% RSLogix 500 project DIAGNOSTICO_ML1400.RSS, saved by version 12.00.00.00 %
PROJECT "UNTITLED"    % processor: type code 64 %

PROGRAM FILES
  LAD 2   15 rungs

DATA FILES
  O0 OUTPUT  6 elements
  I1 INPUT  9 elements
  S2 STATUS  66 elements
  B3 BINARY  1 elements
  T4 TIMER  1 elements
  C5 COUNTER  1 elements
  R6 CONTROL  1 elements
  N7 INTEGER  20 elements
  F8 FLOAT  1 elements

LADDER 2
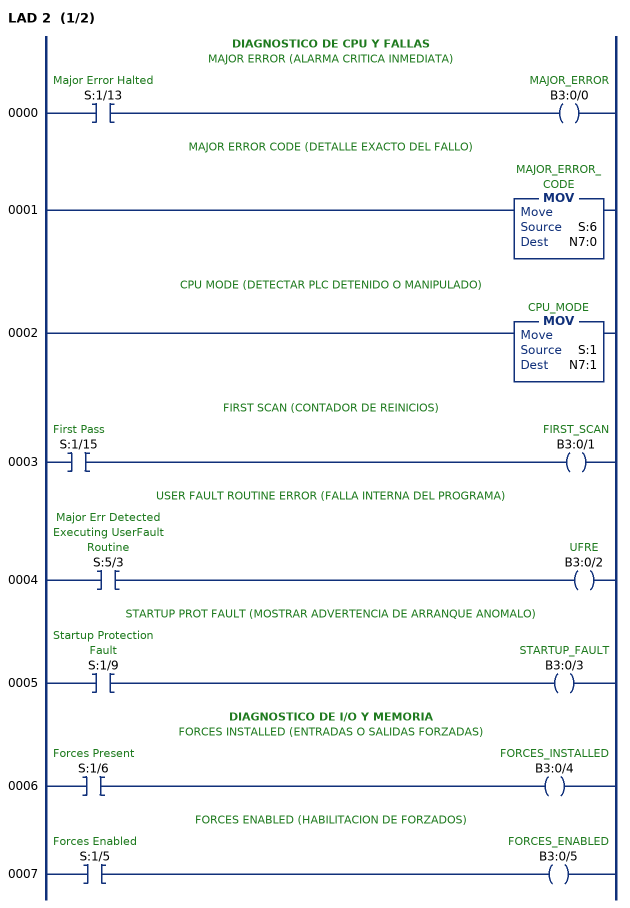
% Rung: 0 %
% TITLE: DIAGNOSTICO DE CPU Y FALLAS %
% MAJOR ERROR (ALARMA CRITICA INMEDIATA) %
SOR XIC S:1/13 OTE B3:0/0 EOR
%   S:1/13  "Major Error Halted" %
%   B3:0/0  MAJOR_ERROR %
% Rung: 1 %
% MAJOR ERROR CODE (DETALLE EXACTO DEL FALLO) %
SOR MOV S:6 N7:0 EOR
%   S:6  "Major Error Fault Code" %
%   N7:0  MAJOR_ERROR_CODE %
% Rung: 2 %
% CPU MODE (DETECTAR PLC DETENIDO O MANIPULADO) %
SOR MOV S:1 N7:1 EOR
%   S:1  "Processor Mode Status/ Control" %
%   N7:1  CPU_MODE %
% Rung: 3 %
% FIRST SCAN (CONTADOR DE REINICIOS) %
SOR XIC S:1/15 OTE B3:0/1 EOR
%   S:1/15  "First Pass" %
%   B3:0/1  FIRST_SCAN %
% Rung: 4 %
% USER FAULT ROUTINE ERROR (FALLA INTERNA DEL PROGRAMA) %
SOR XIC S:5/3 OTE B3:0/2 EOR
%   S:5/3  "Major Err Detected Executing UserFault Routine" %
%   B3:0/2  UFRE %
% Rung: 5 %
% STARTUP PROT FAULT (MOSTRAR ADVERTENCIA DE ARRANQUE ANOMALO) %
SOR XIC S:1/9 OTE B3:0/3 EOR
%   S:1/9  "Startup Protection Fault" %
%   B3:0/3  STARTUP_FAULT %
% Rung: 6 %
% TITLE: DIAGNOSTICO DE I/O Y MEMORIA %
% FORCES INSTALLED (ENTRADAS O SALIDAS FORZADAS) %
SOR XIC S:1/6 OTE B3:0/4 EOR
%   S:1/6  "Forces Present" %
%   B3:0/4  FORCES_INSTALLED %
% Rung: 7 %
% FORCES ENABLED (HABILITACION DE FORZADOS) %
SOR XIC S:1/5 OTE B3:0/5 EOR
%   S:1/5  "Forces Enabled" %
%   B3:0/5  FORCES_ENABLED %

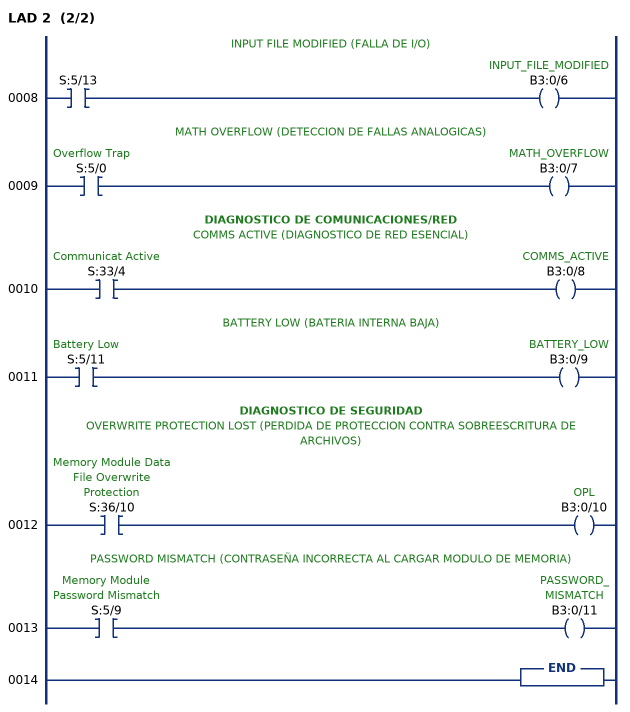
% Rung: 8 %
% INPUT FILE MODIFIED (FALLA DE I/O) %
SOR XIC S:5/13 OTE B3:0/6 EOR
%   B3:0/6  INPUT_FILE_MODIFIED %
% Rung: 9 %
% MATH OVERFLOW (DETECCION DE FALLAS ANALOGICAS) %
SOR XIC S:5/0 OTE B3:0/7 EOR
%   S:5/0  "Overflow Trap" %
%   B3:0/7  MATH_OVERFLOW %
% Rung: 10 %
% TITLE: DIAGNOSTICO DE COMUNICACIONES/RED %
% COMMS ACTIVE (DIAGNOSTICO DE RED ESENCIAL) %
SOR XIC S:33/4 OTE B3:0/8 EOR
%   S:33/4  "Communicat Active" %
%   B3:0/8  COMMS_ACTIVE %
% Rung: 11 %
% BATTERY LOW (BATERIA INTERNA BAJA) %
SOR XIC S:5/11 OTE B3:0/9 EOR
%   S:5/11  "Battery Low" %
%   B3:0/9  BATTERY_LOW %
% Rung: 12 %
% TITLE: DIAGNOSTICO DE SEGURIDAD %
% OVERWRITE PROTECTION LOST (PERDIDA DE PROTECCION CONTRA SOBREESCRITURA DE ARCHIVOS) %
SOR XIC S:36/10 OTE B3:0/10 EOR
%   S:36/10  "Memory Module Data File Overwrite Protection" %
%   B3:0/10  OPL %
% Rung: 13 %
% PASSWORD MISMATCH (CONTRASEÑA INCORRECTA AL CARGAR MODULO DE MEMORIA) %
SOR XIC S:5/9 OTE B3:0/11 EOR
%   S:5/9  "Memory Module Password Mismatch" %
%   B3:0/11  PASSWORD_MISMATCH %
% Rung: 14 %
SOR END EOR

OTHER DOCUMENTED ADDRESSES
  B3:0/12  MODOCPU
  F8:0  MODO_CPU

DATA TABLE (non-zero values as saved)
DATA B3
% B3:0 % 0X0020
DATA N7
% N7:0 % 0 38 0 0 0 0 0 0 0 0
